FUNCTION_BLOCK FB_LongPress
VAR_OUTPUT
	bReset : BOOL;
END_VAR

VAR
	state : INT := 0;
	Button AT%I* : BOOL;
	fbTon : TON := (PT :=T#3S); 
END_VAR

CASE state OF
	0:
		fbTon(IN := FALSE);
		IF Button THEN 
			state := 10;
		END_IF
		
	10:
		fbTon(IN := TRUE);
		IF fbTon.Q THEN 
			IF Button THEN
				bReset := TRUE;
			END_IF
			state := 0;
		END_IF
		IF NOT BUTTON THEN 
			state := 0;
		END_IF
		
END_CASE

END_FUNCTION_BLOCK

(* stored: Version 1.1.0.1, ProductVersion 3.1.4024.12
   POU FB_LongPress: Id {65073088-e608-4819-9920-77a8cf7cacde}, SpecialFunc None *)
